Yaskawa INFORM job: neg_y_0.JBI

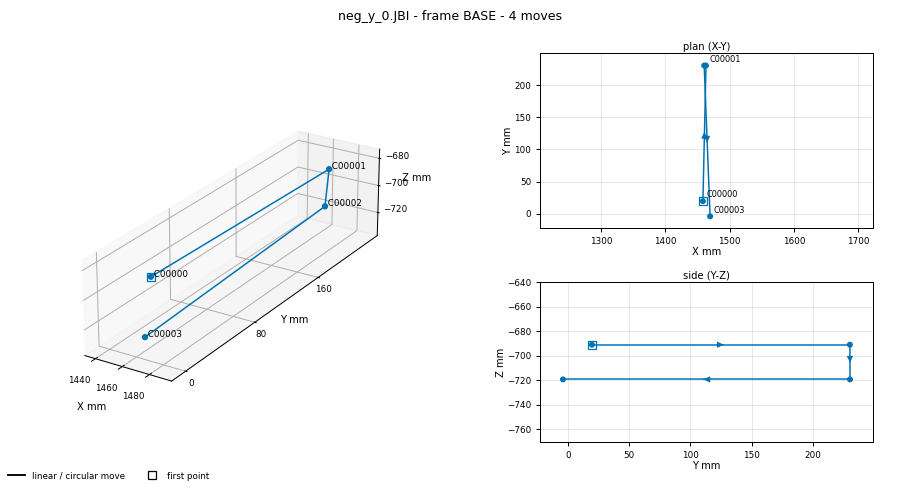
[picture p0: tool path of neg_y_0.JBI in frame BASE, 4 of 6 moves have a stored position in this frame; points joined in program order, loops and branches not executed]
/JOB
//NAME neg_y_0
//POS
///NPOS 4,0,4,0,0,0
///TOOL 0
///POSTYPE BASE
///RECTAN
///RCONF 0,0,0,0,0,0,0,0,0,0,0,0,0,0,0,0,0,0,0,0,0,0,0,0
C00000=1458.453050,19.482825,-691.111355,180.000000,-60.000000,0.000000
C00001=1463.248050,230.242825,-691.111355,180.000000,-60.000000,0.000000
C00002=1460.449050,230.352825,-719.455355,180.000000,-60.000000,0.000000
C00003=1469.614050,-4.187175,-719.455355,180.000000,-60.000000,0.000000
///POSTYPE PULSE
///PULSE
EX000=368640
///POSTYPE PULSE
///PULSE
EC00000=368640
EC00001=368640
EC00002=368640
EC00003=368640
//INST
///DATE 2023/08/07 14:38
///ATTR SC,RW,RJ
////FRAME BASE
///GROUP1 RB1,ST1
NOP
MOVJ P009 EX000 VJ=15.00
MOVJ C00000 EC00000 VJ=15.0
CALL JOB:SPYON
MOVL C00001 EC00001 V=150.0
MOVL C00002 EC00002 V=150.0
MOVL C00003 EC00003 V=150.0
CALL JOB:SPYOF
MOVJ P009 VJ=15.00
END
